INTERFACE I_Event EXTENDS __SYSTEM.IQueryInterface

METHOD PUBLIC AddSubscriber
VAR_INPUT
	Subscriber : I_Subscriber;
END_VAR
END_METHOD

METHOD PUBLIC RemoveSubscriber
VAR_INPUT
	Subscriber : I_Subscriber;
END_VAR
END_METHOD

END_INTERFACE

(* stored: Version 1.1.0.1, ProductVersion 3.1.4024.11
   Itf I_Event: Id {3ef0a490-be40-4d69-8456-a89ecc5f2bc3}
   Method AddSubscriber: Id {df43b343-508b-43eb-a755-7d0e5f4d9ee9}
   Method RemoveSubscriber: Id {a74bacb0-5c6a-408c-a82d-7adb1e93b880} *)
